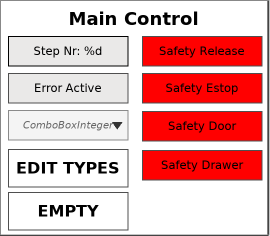
VISUALIZATION vTableState  // 270x236
VAR_IN_OUT
	fbTableControl: FB_TableControl;
END_VAR
    Rectangle (-2,0 270x236)
    Rectangle (8,36 120x30), "Step Nr: %d", text variable: fbTableControl.iWorkStep
    Rectangle (8,73 120x30), "Error Active", colour toggle: fbTableControl.bError
    Rectangle (142,36 120x30), "Safety Release", colour toggle: fbTableControl.bReleaseFromSafety
    Label (61,2 145x34), "Main Control"
    Rectangle (8,149 120x38), "EDIT TYPES"
        OnMouseDown: execute { fbTableControl.stHMI.iDialogNumber:=206; fbTableControl.stHMI.nEditedType:=fbTableControl.stHMI.nCurrentTypeToProduce; }
    ComboBoxInteger (8,110 120x30), variable: fbTableControl.stHMI.nCurrentTypeToProduce, text list: 'tlBottleTypes'
    Rectangle (142,73 120x30), "Safety Estop", colour toggle: fbTableControl.stInOuts.bI_SafetyEstopOK
    Rectangle (142,111 120x30), "Safety Door", colour toggle: fbTableControl.stInOuts.bI_SafetyGateOK
    Rectangle (142,150 120x30), "Safety Drawer", colour toggle: fbTableControl.stInOuts.bI_SafetyDrawerOK
    Rectangle (8,192 120x38), "EMPTY", colour toggle: fbTableControl.stHMI.bEmptyMode
        toggle fbTableControl.stHMI.bEmptyMode
END_VISUALIZATION

(* stored: Version 1.1.0.1, ProductVersion 3.1.4024.15
   Visu vTableState: Id {ffb474ac-bb85-44b3-8906-f3ff8ff9e32e} *)
